# EPICS autosave request: galilDmc30017App/Db/galil_highlevel_settings.req
## High level PVs that should be saved

# Should reset position value to configured Home position
# after a Home procedure?
$(P)RstPosAfterHome-Sel

# Reference Home position value
$(P)RefHomePos-SP

# Backstep tweak to apply after a "homing to limit switch" operation
$(P)HomeToLimSwTweak-SP
